ABB RobotStudio station: Solution_PickAndPlace_SingleRobot.rspag

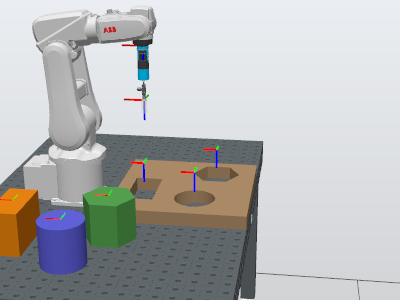
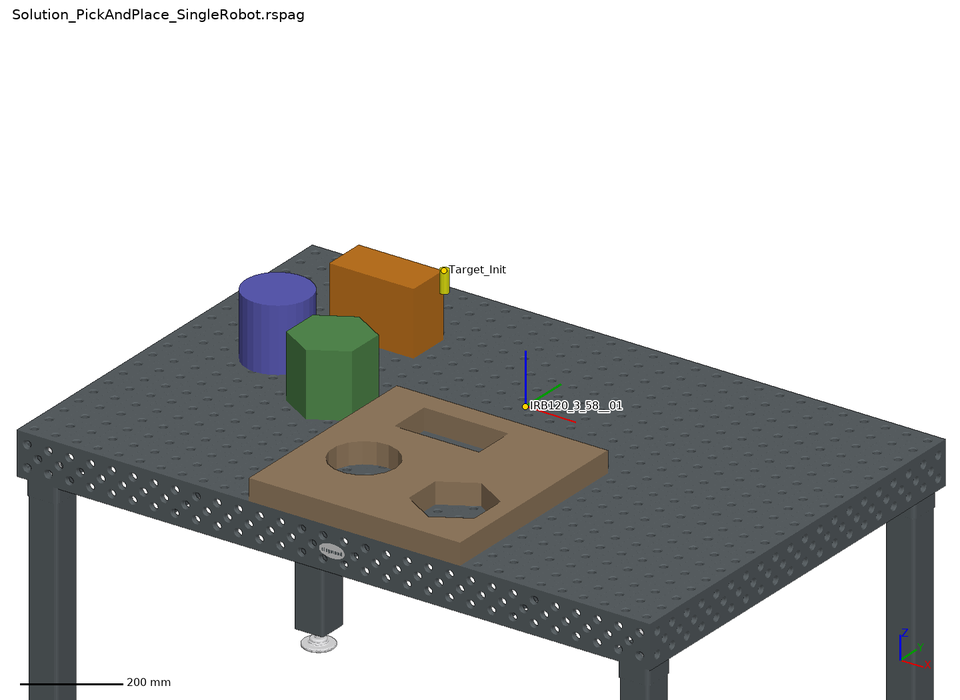
[picture v1: parts stored in the station drawn from their meshes, with robot base, taught points and paths (robot models come from the ABB library and are not in the file)]
--- station ---
Station Solution_1_Tutorial (saved by RobotStudio 22.3.10190.2)
Controller Controller_IRB, task T_ROB1: task frame (RAPID world) sits at (0, 150, 830) mm, rotated rx 0 ry 0 rz -90 deg in the station
Controller Controller_IRB
  mechanical unit ROB_1: IRB120_3_58__01, 6 joints, base frame (0, 0, 0) mm
Layout (positions relative to the parent item):
  - obj_Form [part] at (-200, -500, 830) mm, size 500 x 500 x 50 mm
  - obj_Orange [part] at (-600, -150, 829.97) mm, size 200 x 100 x 150 mm
  - obj_Blue [part] at (-650, -150, 829.56) mm, size 149.5 x 149.7 x 150 mm
  - obj_Green [part] at (-700, -200, 829.84) mm, size 155.5 x 179.5 x 150 mm
  - obj_Table [part], size 1500 x 1010.3 x 830 mm
  - IRB120_3_58__01 [mechanism, from Robots\IRB120_3_58_G_01.rslib] at (0, 150, 830) mm, rotated rx 0 ry 0 rz -90 deg; joint values [-0.0385, -0.1158, -0.0047, 0, 1.6913, -0.0385] (rad or m)
  - smc_Gripper [mechanism, from Gripper_RS_tool\smc_gripper.rslib] at (-10, -110, 1422) mm, rotated rx 180 ry 0 rz 90 deg
  - LineSensor [smart component, from Components\LineSensor.rslib] at (-10, -110, 1228.31) mm, rotated rx 180 ry 0 rz 90 deg
      properties: Start=[0 0 0]; End=[-4.8722724414231E-07 4.44425481930123E-16 0.0500000031816989]; Radius=0.01; SensedPart=(none); SensedPoint=[0 0 0]
    - _sensorPart_ [part], size 20 x 20 x 50 mm
  - Attacher [smart component, from Components\Attacher.rslib]
      properties: Parent=smc_Gripper; Flange=0; Child=(none); Mount=false; Offset=[0 0 0]; Orientation=[0 0 0]
  - Detacher [smart component, from Components\Detacher.rslib]
      properties: Child=(none); KeepPosition=true
  - Part_3 [part]
Attachment: smc_Gripper is attached to IRB120_3_58__01 / Link6
Attachment: LineSensor is attached to smc_Gripper / Assembly_ABBGRIP_2
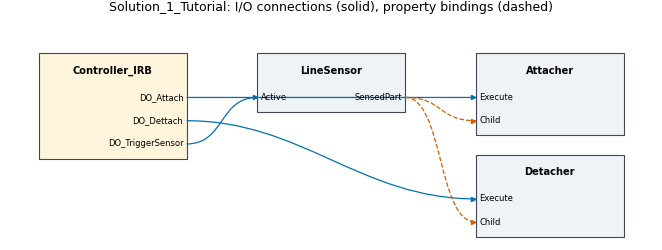
Station logic (signal -> signal, property => property):
  Controller_IRB.DO_Attach -> Attacher.Execute
  Controller_IRB.DO_Dettach -> Detacher.Execute
  Controller_IRB.DO_TriggerSensor -> LineSensor.Active
  LineSensor.SensedPart => Attacher.Child
  LineSensor.SensedPart => Detacher.Child

--- Backups/Controller_IRB/RAPID/TASK1/PROGMOD/CalibData.mod ---
MODULE CalibData
    PERS tooldata smc_gripper:=[TRUE,[[0,0.004,197.001],[1,0,0,0]],[1,[0.207,-0.496,71.18],[1,0,0,0],0,0,0]];
ENDMODULE

--- Backups/Controller_IRB/RAPID/TASK1/PROGMOD/Module1.mod ---
MODULE Module1
    CONST robtarget Target_Init:=[[260,-10,395],[-0.000000095,0,1,0],[-1,-1,-1,0],[9E+09,9E+09,9E+09,9E+09,9E+09,9E+09]];
    CONST robtarget Target_PickBlue:=[[100,-517.298,150],[-0.000000095,0,1,0],[0,0,0,0],[9E+09,9E+09,9E+09,9E+09,9E+09,9E+09]];
    CONST robtarget Target_PlaceBlue:=[[450,-67.298,150],[-0.000000095,0,1,0],[0,0,0,0],[9E+09,9E+09,9E+09,9E+09,9E+09,9E+09]];
    CONST robtarget Target_PickGreen:=[[200,-317.298,150],[-0.000000095,0,1,0],[0,0,0,0],[9E+09,9E+09,9E+09,9E+09,9E+09,9E+09]];
    CONST robtarget Target_PlaceGreen:=[[500,182.702,150],[-0.000000095,0,1,0],[0,0,0,0],[9E+09,9E+09,9E+09,9E+09,9E+09,9E+09]];
    CONST robtarget Target_PickOrange:=[[-100,-400,150],[-0.000000095,0,1,0],[0,0,0,0],[9E+09,9E+09,9E+09,9E+09,9E+09,9E+09]];
    CONST robtarget Target_PlaceOrange:=[[250,0,150],[-0.000000095,0,1,0],[0,0,0,0],[9E+09,9E+09,9E+09,9E+09,9E+09,9E+09]];

    CONST num PICK_OFFSET:=50;
    CONST num SAFE_OFFSET:=80;
    !***********************************************************
    !
    ! Module:  Module_PickAndPlaceRoutine
    !
    ! Description:
    !   Simple pick-and-place task is performed by IRB
    !
    ! Author: Egor Ch.
    !
    ! Version: 1.0
    !
    !***********************************************************
    PROC main()
        PickPlaceToForm Target_PickGreen,Target_PlaceGreen;
        PickPlaceToForm Target_PickBlue,Target_PlaceBlue;
        PickPlaceToForm Target_PickOrange,Target_PlaceOrange;
        PickPlaceToForm Target_PlaceOrange,Target_PickOrange;
        PickPlaceToForm Target_PlaceBlue,Target_PickBlue;
        PickPlaceToForm Target_PlaceGreen,Target_PickGreen;
    ENDPROC

    PROC PickPlaceToForm(robtarget Target_Pick,robtarget Target_Place)
        SetDO DO_TriggerSensor,1;
        SetDO DO_Dettach,1;
        WaitTime 0.2;
        SetDO DO_Dettach,0;
        SetDO DO_TriggerSensor,0;

        MoveL Target_Init,v1000,fine,smc_gripper\WObj:=wobj0;

        MoveL Offs(Target_Pick,0,0,PICK_OFFSET),v1000,z20,smc_gripper\WObj:=wobj0;
        MoveL Target_Pick,v1000,fine,smc_gripper\WObj:=wobj0;

        SetDO DO_TriggerSensor,1;
        SetDO DO_Attach,1;
        WaitTime 0.5;
        SetDO DO_TriggerSensor,0;

        MoveL Offs(Target_Pick,0,0,SAFE_OFFSET),v1000,z20,smc_gripper\WObj:=wobj0;

        MoveL Offs(Target_Place,0,0,PICK_OFFSET),v1000,fine,smc_gripper\WObj:=wobj0;
        MoveL Target_Place,v1000,fine,smc_gripper\WObj:=wobj0;

        SetDO DO_TriggerSensor,1;
        SetDO DO_Attach,0;
        SetDO DO_Dettach,1;
        WaitTime 0.2;
        SetDO DO_Dettach,0;
        SetDO DO_TriggerSensor,0;

        MoveL Target_Init,v1000,fine,smc_gripper\WObj:=wobj0;
    ENDPROC
ENDMODULE

--- Backups/Controller_IRB/SYSPAR/EIO.cfg ---
EIO:CFG_1.0:6:1::
#
EIO_SIGNAL:

      -Name "DO_Attach" -SignalType "DO"

      -Name "DO_Dettach" -SignalType "DO"

      -Name "DO_TriggerSensor" -SignalType "DO"
